FUNCTION TryConvert_BOOL_TO_BYTE : BOOL
VAR_INPUT
	in : BOOL;
	out : REFERENCE TO BYTE;
END_VAR

out := BOOL_TO_BYTE(in);
TryConvert_BOOL_TO_BYTE := TRUE;

END_FUNCTION

(* stored: Version 1.1.0.1, ProductVersion 3.1.4024.12
   POU TryConvert_BOOL_TO_BYTE: Id {64563b63-f711-4b59-a926-4ff42225720c}, SpecialFunc None *)
